FUNCTION_BLOCK BigDemux (* Basic Function Block Type *)
  (* Standard: 61499-2 *)
  (* Version 0.0, 6/8/2016, Andrei, nxtControl GmbH, Template *)
  PACKAGE Main;
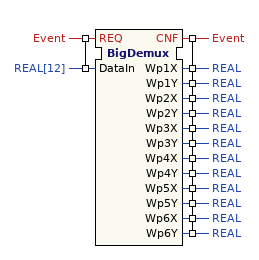
  EVENT_INPUT
    REQ WITH DataIn; (* Normal Execution Request *)
  END_EVENT
  EVENT_OUTPUT
    CNF WITH Wp1X, Wp1Y, Wp2X, Wp2Y, Wp3X, Wp3Y, Wp4X, Wp4Y, Wp5X, Wp5Y, Wp6X, Wp6Y; (* Execution Confirmation *)
  END_EVENT
  VAR_INPUT
    DataIn : ARRAY [0..11] OF REAL; (* Input event qualifier *)
  END_VAR
  VAR_OUTPUT
    Wp1X : REAL; (* Output event qualifier *)
    Wp1Y : REAL;
    Wp2X : REAL;
    Wp2Y : REAL;
    Wp3X : REAL;
    Wp3Y : REAL;
    Wp4X : REAL;
    Wp4Y : REAL;
    Wp5X : REAL;
    Wp5Y : REAL;
    Wp6X : REAL;
    Wp6Y : REAL;
  END_VAR
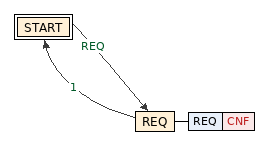
  EC_STATES
    START; (* Initial State *)
    REQ : REQ -> CNF; (* Normal execution *)
  END_STATES
  EC_TRANSITIONS
    START TO REQ := REQ;
    REQ TO START := 1;
  END_TRANSITIONS
  ALGORITHM REQ IN ST: (* Normally executed algorithm *)
Wp1X := DataIn[0];
Wp1Y := DataIn[1];
Wp2X := DataIn[2];
Wp2Y := DataIn[3];
Wp3X := DataIn[4];
Wp3Y := DataIn[5];
Wp4X := DataIn[6];
Wp4Y := DataIn[7];
Wp5X := DataIn[8];
Wp5Y := DataIn[9];
Wp6X := DataIn[10];
Wp6Y := DataIn[11];
  END_ALGORITHM
END_FUNCTION_BLOCK
